ABB RobotStudio station: SolutioneditTEST02.rspag

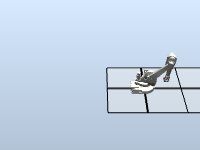
--- station ---
Station Solution149 (saved by RobotStudio 6.6.7701.1025)
Controller 1600-514385
  mechanical unit ROB_1: IRB1600_10_145__01, 6 joints, base frame (0, 0, 0) mm
Layout (positions relative to the parent item):
  - IRB1600_10_145__01 [mechanism, from Robots\IRB1600_10_145_G_01.rslib] at (0, 0, 0) mm; joint values [-0.2814, 0.7661, 0.9215, 1.2913, 1.5384, -1.683] (rad or m)

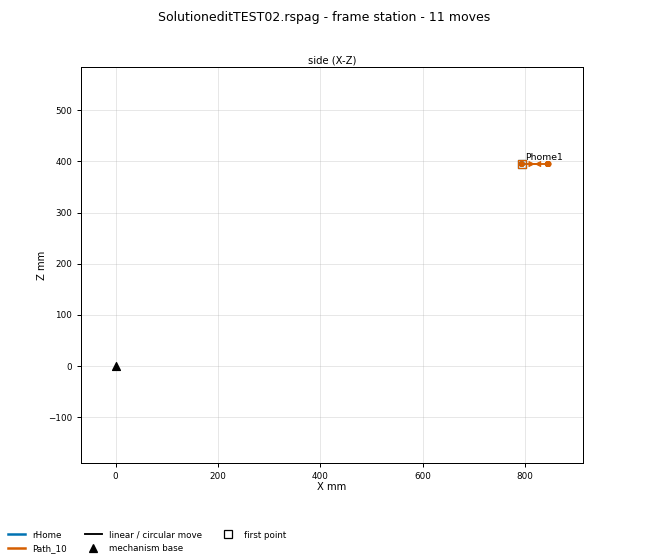
[picture p0: tool path of SolutioneditTEST02.rspag in frame station, 11 of 11 moves have a stored position in this frame; points joined in program order, loops and branches not executed]
--- Backups/1600-514385/RAPID/TASK1/PROGMOD/CalibData.mod ---
MODULE CalibData





ENDMODULE

--- Backups/1600-514385/RAPID/TASK1/PROGMOD/MainModule.mod ---
MODULE MainModule

    CONST robtarget Phome1:=[[-220,250,60],[0.5,0.5,0.5,0.5],[-1,0,-2,0],[9E+09,9E+09,9E+09,9E+09,9E+09,9E+09]];
    CONST robtarget Phome2:=[[-185,250,60],[0.5,0.5,0.5,0.5],[-1,0,-2,0],[9E+09,9E+09,9E+09,9E+09,9E+09,9E+09]];

	PROC main()
		Path_10;
!        rHome;

	ENDPROC
	PROC rHome()
		MoveL Phome1,v100,z50,Polish0101\WObj:=Workobject_1;
	ENDPROC

ENDMODULE

--- Backups/1600-514385/RAPID/TASK1/PROGMOD/Module1.mod ---
MODULE Module1

    VAR speeddata vx1:=[114/1,10,1,1];
    VAR speeddata vx2:=[114/2,10,1,1];
    VAR speeddata vx3:=[114/3,10,1,1];
    VAR speeddata vx4:=[114/4,10,1,1];
    VAR speeddata vx5:=[114/5,10,1,1];
  PERS tooldata Polish0101:=[TRUE,[[-251,0,89],[0.707107,0,-0.707107,0]],[8.4,[65,0,90],[1,0,0,0],0,0,0]];
  PERS wobjdata Workobject_1:=[FALSE,TRUE,"",[[1014.2,-253,335],[1,0,0,0]],[[0,0,0],[1,0,0,0]]];


  PERS num Cycle_num:=2;
  PERS num numsp;
!     frame.trans:=[50,0,40];

  PERS pose f:=[[10,15,10],[1,0.5,0,0]];

	CONST robtarget Target_10:=[[-169.2,250.000000051,60],[0.49914225,0.49914225,0.500856281,0.500856281],[-1,0,-2,0],[9E+09,9E+09,9E+09,9E+09,9E+09,9E+09]];
	CONST robtarget Target_20:=[[-169.095154964,250.992581655,60],[0.549643456,0.549643456,0.444850617,0.444850617],[-1,1,-2,0],[9E+09,9E+09,9E+09,9E+09,9E+09,9E+09]];
	CONST robtarget Target_30:=[[-168.793229078,251.944319114,60],[0.58959812,0.58959812,0.390351197,0.390351197],[-1,1,-2,0],[9E+09,9E+09,9E+09,9E+09,9E+09,9E+09]];
	CONST robtarget Target_40:=[[-168.323393963,252.8256452,60],[0.621207026,0.621207026,0.337789626,0.337789626],[0,1,-2,0],[9E+09,9E+09,9E+09,9E+09,9E+09,9E+09]];
	CONST robtarget Target_50:=[[-167.718295046,253.620660361,60],[0.644380732,0.644380732,0.291158844,0.291158844],[0,1,-2,0],[9E+09,9E+09,9E+09,9E+09,9E+09,9E+09]];
	PROC Path_10()
	    MoveL Phome1,v100,fine,Polish0101\WObj:=Workobject_1;
        numsp:=0;
        FOR n FROM 1 TO Cycle_num DO
        MoveL Target_10,vx1,z20,Polish0101\WObj:=Workobject_1;
	    MoveL Target_20,vx2,z20,Polish0101\WObj:=Workobject_1;
	    MoveL Target_30,vx3,z20,Polish0101\WObj:=Workobject_1;
	    MoveL Target_40,vx4,z20,Polish0101\WObj:=Workobject_1;
	    MoveL Target_50,vx5,fine,Polish0101\WObj:=Workobject_1;
	    MoveL Target_40,vx4,z20,Polish0101\WObj:=Workobject_1;
	    MoveL Target_30,vx3,z20,Polish0101\WObj:=Workobject_1;
        MoveL Target_20,vx2,fine,Polish0101\WObj:=Workobject_1;
        numsp:=numsp+1;
        ENDFOR
!
         MoveL Phome1,v100,z50,Polish0101\WObj:=Workobject_1;
	ENDPROC
ENDMODULE

--- Backups/1600-514385/RAPID/TASK1/SYSMOD/LINKEDM.sys ---
%%%
  VERSION:1
  LANGUAGE:ENGLISH
%%%

MODULE LINKEDM (SYSMODULE)

! FOLLOWER
!     Name of electronically linked follower axis used by operator at teach pendent.
      PERS string l_f_axis_name{5}       :=  ["",  "", "", "", ""];

!     Name of the mechanical unit for follower axis.
      PERS string l_f_mecunt_n{5}  :=  ["", "", "", "", ""];

!     Linked follower axis number in the mechanical unit (first axis in mech. unit is number 1).
      PERS num l_f_axis_no{5}      :=  [0,          0,   0,  0,  0];

! MASTER
!     Name of the mechanical unit for linked master axis.
      PERS string l_m_mecunt_n{5} :=  ["", "", "", "", ""];

!     Linked master axis number in the mechanical unit (first axis in mech. unit is number 1).
!     See axis number table in documentation for different master mechanical units.
      PERS num l_m_axis_no{5}     :=  [0,  0,  0,  0,  0];

! POSITION OFFSET
!     The increase of the allowed offset position between the master and follower
!     positions, used when starting AUTO mode. As soon as the offset is decreased
!     the old configurated parameter is used.
!     Example: 3 => the configurated value of allowed offset is increased 3 times.
      PERS num offset_ratio{5}       :=  [10,  10,   10,  10,  10];

! SPEED RATIO
!     Speed_ratio used in AUTO and JOG modes [ very_slow   slow    normal    fast]
!     Value 1 = max allowed manual speed.
      CONST num speed_ratio {20}      := [0.01, 0.01, 0.01, 0.01, 0.01,
                                          0.05, 0.05, 0.05, 0.05, 0.05,
                                          0.20, 0.20, 0.20, 0.20, 0.20,
                                          1.00, 1.00, 1.00, 1.00, 1.00];

! STEP SIZE
!     Displacement position used in JOG mode for each activation of positive or
!     negative movement.                  [very_short    short   normal   long]
!     Unit degees or meter.
      CONST num displacement {20}     := [0.001, 0.001, 0.001, 0.001, 0.001,
                                          0.005, 0.005, 0.005, 0.005, 0.005,
                                          0.020, 0.020, 0.020, 0.020, 0.020,
                                          0.100, 0.100, 0.100, 0.100, 0.100];


!-------------------------------------------------------------
 PROC Linked_m ()
      Linked_m_exe ;
 ENDPROC
ENDMODULE

--- Backups/1600-514385/SYSPAR/EIO.cfg ---
EIO:CFG_1.0:6:1::
#
INDUSTRIAL_NETWORK:

      -Name "DeviceNet" -Label "DeviceNet Master/Slave Network" -Address "2"
#
DEVICENET_INTERNAL_DEVICE:

      -Name "DN_Internal_Device" -VendorName "ABB Robotics"\
      -ProductName "DeviceNet Internal Slave Device"
